{attribute 'GeneratedUsingTerminal: EL9184--0000'}
{attribute addProperty BoxType "EL9184--0000"}
{attribute addProperty Description "EL9184 Potential Connection, 8 x 24V, 8 x Ground"}
{attribute addProperty Physics "KK"}
{attribute addProperty Id "EL9184"}
{attribute addProperty CRC "2551281744"}
{attribute addProperty Size "0"}
TYPE EL9184_98117850 EXTENDS EtcSlaveTerminalBase_947E5A46 :
STRUCT
END_STRUCT
END_TYPE

(* stored: Version 1.2.0.0, ProductVersion 3.1.4024.11
   DUT EL9184_98117850: Id {97010b1c-7d67-4ae2-8a2d-2df65de8f8f0} *)
